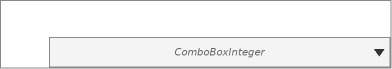
VISUALIZATION Taschenrechner  // 392x69
    ComboBoxInteger (49,37 341x30), variable: MAIN.TaschenRechner.Befehl, text list: 'TaschenrechnerBefehle'
END_VISUALIZATION

(* stored: Version 1.1.0.1, ProductVersion 3.1.4022.6
   Visu Taschenrechner: Id {529ab607-a3a7-4016-be48-cafee3caa910} *)
